FUNCTION_BLOCK PostVentilation
VAR_INPUT
	EN: BOOL := TRUE;
	SP: LREAL;
	PostVentilationTime: LTIME := LTIME#2M;
	PostVentilationLevel: LREAL := 0.25;
END_VAR
VAR_OUTPUT
	ENO: BOOL;
	SP_PostVentilation: LREAL;
END_VAR
VAR
	PostVentilationTOF: TOF;
END_VAR

PostVentilationTOF(IN := SP > 0.01, PT := LTIME_TO_TIME(PostVentilationTime));
IF EN THEN
	IF PostVentilationTOF.Q THEN
		ENO := TRUE;
		IF SP > 0.01 THEN
			SP_PostVentilation := SP;
		ELSE
			SP_PostVentilation := PostVentilationLevel;
		END_IF
	ELSE
		ENO := FALSE;
		SP_PostVentilation := 0;
	END_IF
ELSE
	ENO := FALSE;
	SP_PostVentilation := SP;
END_IF

END_FUNCTION_BLOCK

(* stored: Version 1.1.0.1, ProductVersion 3.1.4024.6
   POU PostVentilation: Id {8d656c1b-4d9d-4f1a-a51c-c8e5edc13b2d}, SpecialFunc None *)
